FUNCTION UpdateLogTimestampWithSystemTime
VAR_INPUT
	stEvent : REFERENCE TO  ST_LogEntry;
END_VAR
VAR
	fbGETSYSTEMTYPE : GETSYSTEMTIME;
	stFileTime : T_FILETIME;
END_VAR

fbGETSYSTEMTYPE(timeLoDW => stFileTime.dwLowDateTime, 
				timeHiDW =>  stFileTime.dwHighDateTime);
				
stEvent.dtTimestamp := FILETIME_TO_DT(fileTime := stFileTime);

END_FUNCTION

(* stored: Version 1.1.0.1
   POU UpdateLogTimestampWithSystemTime: Id {9b2b7fed-42ab-4ae9-be5d-c53f4111b5db}, SpecialFunc None *)
